// TIA Portal project "datadiode_sender_v2" (V17)

(* hardware
DEVICE "S7-1500/ET200MP-Station_1"  S7-1500 station
   slot 0: "Profilschiene_0"  Rack  6ES7 590-1***0-0AA0
   slot 1: "PLC_1"  CPU 1516-3 PN/DP  6ES7 516-3AN02-0AB0  V2.9
      slot 3: "CPU-Display_1"  6ES7591-1BA00-0AA0
      slot 32768: "PROFINET-Schnittstelle_1"  X1
      slot 33024: "PROFINET-Schnittstelle_2"  X2
      slot 33280: "DP-Schnittstelle_1"  X3
      slot 34817: "Virtual CP interface port_1"  Virtual CP interface port  Virtual CP interface port
DEVICE "S7-1500/ET200MP-Station_2"  S7-1500 station
   slot 0: "Profilschiene_0"  Rack  6ES7 590-1***0-0AA0
   slot 1: "workstation4.rio"  IM 155-5 PN ST  6ES7 155-5AA01-0AB0  V4.1
   slot 2: "DI 32x24VDC HF_1"  DI 32x24VDC HF  6ES7 521-1BL00-0AB0  V2.0
   slot 3: "DQ 32x24VDC/0.5A HF_1"  DQ 32x24VDC/0.5A HF  6ES7 522-1BL01-0AB0  V1.0
   slot 4: "AI 8xU/I/RTD/TC ST_1"  AI 8xU/I/RTD/TC ST  6ES7 531-7KF00-0AB0  V2.0
   slot 5: "AQ 8xU/I HS_1"  AQ 8xU/I HS  6ES7 532-5HF00-0AB0  V2.0
DEVICE "GSD-Geraet_1"  GSD.Device.PN
   slot 0: "Baugruppenträger"  Rack  V1.0
   slot 0: "datadiodesender"  Datadiodesender  123 444 555  V0.1.0
      slot 0: "Datadiodesender"  Datadiodesender
      slot 1: "X1"  X1
         slot 1: "X1 P1"  X1 P1
      slot 1: "Status module_1"  Status module  1.0
         slot 0: "Status Submodule"  Status Submodule
   slot 2: "Temperature Module_1"  Temperature Module  1.0
      slot 0: "Temperature submodule"  Temperature submodule
   slot 3: "Tank Module_1"  Tank Module  1.0
      slot 0: "tank submodule"  tank submodule
   slot 4: "Flow rate Module_1"  Flow rate Module  1.0
      slot 0: "Flow rate Submodule"  Flow rate Submodule
   slot 5: "Pressure Module_1"  Pressure Module  1.0
      slot 0: "Pressure Submodule"  Pressure Submodule
*)

// ===== PLC "PLC_1"  CPU 1516-3 PN/DP =====

VAR_GLOBAL   // PLC tag table "Standard-Variablentabelle"
   "TemperatureButton" AT %I0.0 : Bool;
   "TankButton" AT %I0.1 : Bool;
   "FlowRateButton" AT %I0.2 : Bool;
   "TemperatureLED" AT %Q0.0 : Bool;
   "TankLED" AT %Q0.1 : Bool;
   "FlowRateLED" AT %Q0.2 : Bool;
   "PressureLED" AT %Q0.3 : Bool;
   "StatusV" AT %QW20 : UInt;
   "TempV" AT %QW22 : UInt;
   "TankV" AT %QW24 : UInt;
   "FlowrateV" AT %QD26 : Real;
   "PressureV" AT %QD30 : Real;
END_VAR

ORGANIZATION_BLOCK "Main"   // OB1, LAD, ProgramCycle
TITLE = "Main Program Sweep (Cycle)"
{ S7_Optimized_Access := 'TRUE' }
VERSION : 0.1
   VAR_INPUT
      Initial_Call : Bool;   // Initial call of this OB
      Remanence : Bool;   // =True, if remanent data are available
   END_VAR
   VAR CONSTANT
      status_const : UInt := 1;
      temp_const : UInt := 123;
      tank_const : UInt := 300;
      flowrate_const : Real := 40.33;
      pressure_const : Real := 1023.87;
   END_VAR
BEGIN

REGION Network 1
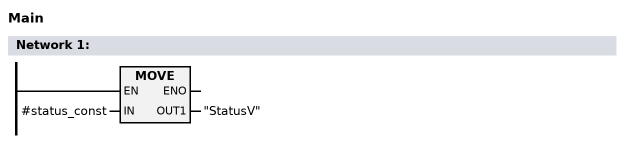
   RUNG wire#powerrail
      Move(in := #status_const, out1 => "StatusV")
   END_RUNG
   // the same network as SCL:
   "StatusV" := #status_const;
END_REGION

REGION Network 2 (SCL)
   IF "TemperatureButton" AND NOT "TankButton" THEN
       "TempV" := #temp_const;
       "TemperatureLED" := TRUE;
   ELSE
       "TempV" := 0;
       "TemperatureLED" := FALSE;
   END_IF;
END_REGION

REGION Network 3 (SCL)
   IF "TankButton" AND NOT "TemperatureButton" THEN
       "TankV" := #tank_const;
       "TankLED" := TRUE;
   ELSE
       "TankV" := 0;
       "TankLED" := false;
   END_IF;
END_REGION

REGION Network 4 (SCL)
   IF "FlowRateButton" THEN
       "FlowrateV" := #flowrate_const;
       "FlowRateLED" := TRUE;
   ELSE
       "FlowrateV" := 0;
       "FlowRateLED" := FALSE;
   END_IF;
END_REGION

REGION Network 5 (SCL)
   IF "TemperatureButton" AND "TankButton" THEN
       "PressureV" := #pressure_const;
       "PressureLED" := TRUE;
   ELSE
       "PressureV" := 0;
       "PressureLED" := FALSE;
   END_IF;
END_REGION
END_ORGANIZATION_BLOCK